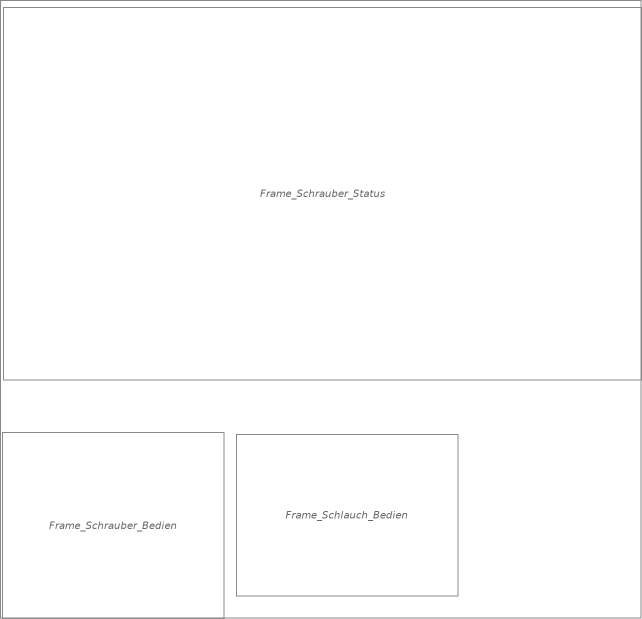
VISUALIZATION Frame_Schrauber  // 642x619
VAR_IN_OUT
	stSKSSchrauberInOut	:ST_SKSSchrauberInOut_Vis;
END_VAR
    Frame (236,434 222x162)
        shows Frame_Schlauch_Bedien(bSchlauchBelegt := stSKSSchrauberInOut.I_bSchlauchBelegt, bSchrauberBelegt := stSKSSchrauberInOut.I_bSchrauberBelegt, bAuswurfStart := stSKSSchrauberInOut.I_bAuswurfStart)
    Frame (2,432 222x187)
        shows Frame_Schrauber_Bedien(bTaktFreigabe := stSKSSchrauberInOut.I_bTaktFrg, bTaktStart := stSKSSchrauberInOut.I_bTaktStart, bTaktStop := stSKSSchrauberInOut.I_bTaktStop, bQuitError := stSKSSchrauberInOut.I_bQuittFehler)
    Frame (3,7 639x373)
        shows Frame_Schrauber_Status(sState := stSKSSchrauberInOut.Q_sStatus, bGrdstlgSchrEinh := stSKSSchrauberInOut.I_bGrdstlgSchrEinh, bZustellZylAusgef := stSKSSchrauberInOut.I_bZustellZylAusgef, bBusy := stSKSSchrauberInOut.Q_bBusy, bDone := stSKSSchrauberInOut.Q_bDone, bError := stSKSSchrauberInOut.Q_bError, bErrorDrehmoment := stSKSSchrauberInOut.Q_bDrehmomentFehler, bDrehmomentOk := stSKSSchrauberInOut.Q_bDrehmomentOk, nDrehmomentMw := stSKSSchrauberInOut.Q_nActTorque, nActPos := stSKSSchrauberInOut.Q_nActPos, nActVelo := stSKSSchrauberInOut.Q_nActVelo, nActTiefe := stSKSSchrauberInOut.Q_nActDepth, nDrehmomentLetzteSchr := stSKSSchrauberInOut.Q_nLastTorque, nTiefeLetzteSchr := stSKSSchrauberInOut.Q_nLastDepth)
END_VISUALIZATION

(* stored: Version 1.1.0.1, ProductVersion 3.1.4024.15
   Visu Frame_Schrauber: Id {d8d56547-8dfc-461d-83ed-f13692911c17} *)
